FUNCTION_BLOCK FB_CTD (* Down counter *)
  (* Standard: 61499-1; Description: Copyright (c) 2023 Martin Erich Jobst This program and the accompanying materials are made available under the terms of the Eclipse Public License 2.0 which is available at https://www.eclipse.org/legal/epl-2.0/ SPDX-License-Identifier: EPL-2.0 *)
  (* Version 1.0, 2023-04-28, Martin Jobst *)
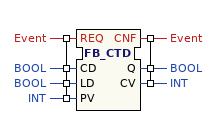
  EVENT_INPUT
    REQ WITH CD, PV, LD; (* Normal Execution Request *)
  END_EVENT
  EVENT_OUTPUT
    CNF WITH Q, CV; (* Execution Confirmation *)
  END_EVENT
  VAR_INPUT
    CD : BOOL; (* Count down *)
    LD : BOOL; (* Load *)
    PV : INT; (* Preset value *)
  END_VAR
  VAR_OUTPUT
    Q : BOOL; (* Output *)
    CV : INT; (* Count value *)
  END_VAR
  ALGORITHM REQ IN ST:
IF LD THEN
  CV := PV;
ELSIF CD AND CV > -32768 THEN
  CV := CV - 1;
END_IF;
Q := CV <= 0;
  END_ALGORITHM
END_FUNCTION_BLOCK
